// Mitsubishi GX Works2 project: project_main   PLC: Q02U

PROGRAM INPUT
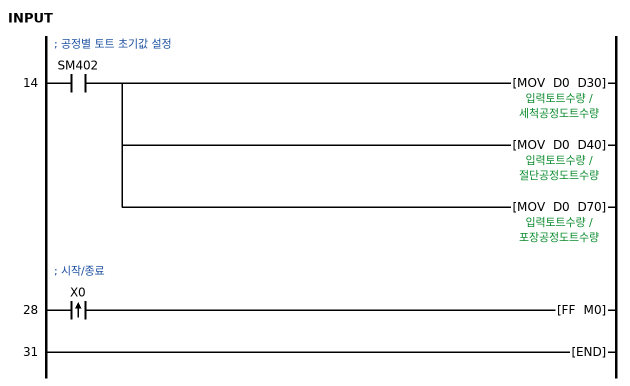
; 공정별 토트 초기값 설정
14    LD      SM402
      MOV     D0 D30  ; 입력토트수량 / 세척공정도트수량
      MOV     D0 D40  ; 절단공정도트수량
      MOV     D0 D70  ; 포장공정도트수량
; 시작/종료
28    LDP     X0
      FF      M0
31    END
END_PROGRAM

PROGRAM 세척공정
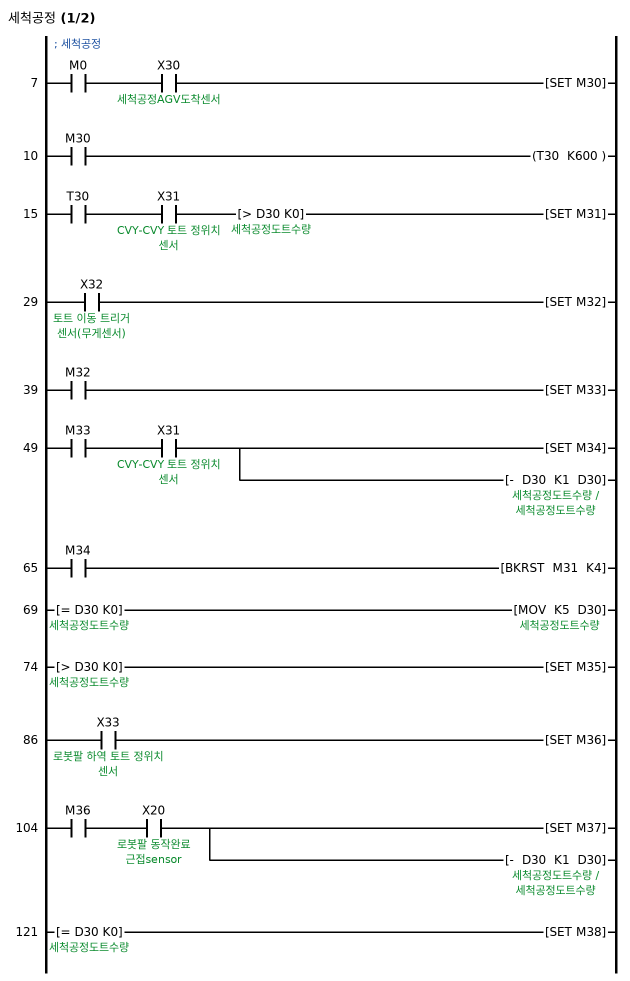
; 세척공정
7     LD      M0
      AND     X30  ; 세척공정AGV도착센서
      SET     M30
10    LD      M30
      OUT     T30 K600
15    LD      T30
      AND     X31  ; CVY-CVY 토트 정위치 센서
      AND>    D30 K0  ; 세척공정도트수량
      SET     M31
        [note] MainCVY ON
29    LD      X32  ; 토트 이동 트리거 센서(무게센서)
      SET     M32
        [note] MAinCVY OFF
39    LD      M32
      SET     M33
        [note] SubCVY1,2 ON
49    LD      M33
      AND     X31  ; CVY-CVY 토트 정위치 센서
      SET     M34
        [note] SubCVY1,2 OFF
      -       D30 K1 D30
65    LD      M34
      BKRST   M31 K4
69    LD=     D30 K0  ; 세척공정도트수량
      MOV     K5 D30
74    LD>     D30 K0  ; 세척공정도트수량
      SET     M35
        [note] SubCVY2 ON
86    LD      X33  ; 로봇팔 하역 토트 정위치 센서
      SET     M36
        [note] SubCVY2 OFF, 하역 로봇팔 ON
104   LD      M36
      AND     X20  ; 로봇팔 동작완료 근접sensor
      SET     M37
        [note] 하역 로봇팔 OFF
      -       D30 K1 D30
121   LD=     D30 K0  ; 세척공정도트수량
      SET     M38
        [note] AGV 다음 공정 이동
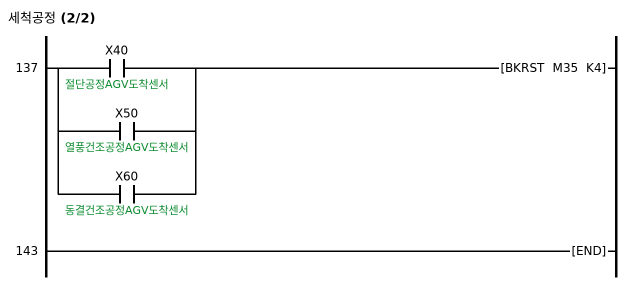
137   LD      X40  ; 절단공정AGV도착센서
      OR      X50  ; 열풍건조공정AGV도착센서
      OR      X60  ; 동결건조공정AGV도착센서
      BKRST   M35 K4
143   END
END_PROGRAM

PROGRAM 열풍건조
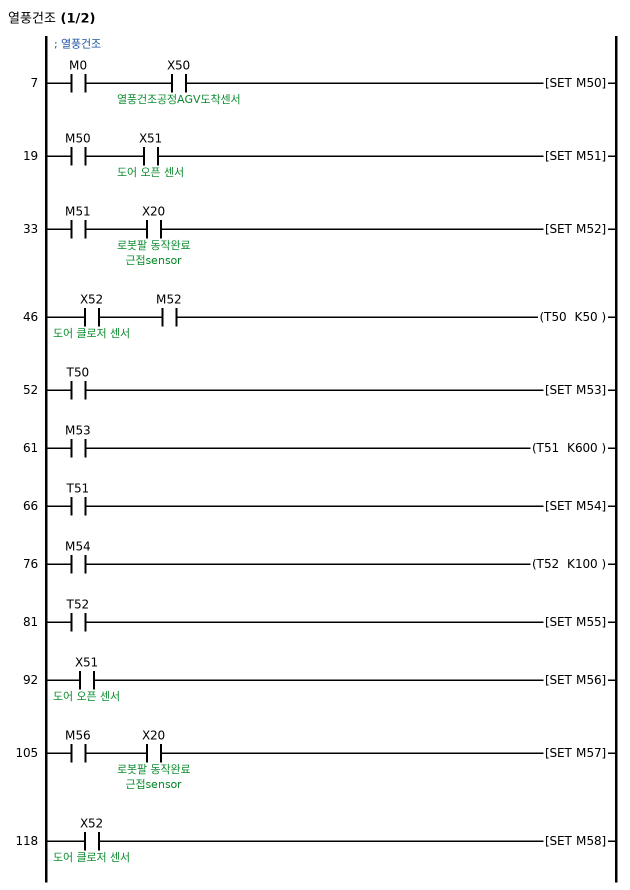
; 열풍건조
7     LD      M0
      AND     X50  ; 열풍건조공정AGV도착센서
      SET     M50
        [note] 도어 오픈CLY
19    LD      M50
      AND     X51  ; 도어 오픈 센서
      SET     M51
        [note] 상역 로봇 팔동작
33    LD      M51
      AND     X20  ; 로봇팔 동작완료 근접sensor
      SET     M52
        [note] 도어 클로즈CYL
46    LD      X52  ; 도어 클로저 센서
      AND     M52
      OUT     T50 K50
52    LD      T50
      SET     M53
        [note] 건조기 ON
61    LD      M53
      OUT     T51 K600
66    LD      T51
      SET     M54
        [note] 건조기 OFF
76    LD      M54
      OUT     T52 K100
81    LD      T52
      SET     M55
        [note] 도어 오픈CYL
92    LD      X51  ; 도어 오픈 센서
      SET     M56
        [note] 하역 로봇팔 동작
105   LD      M56
      AND     X20  ; 로봇팔 동작완료 근접sensor
      SET     M57
        [note] 도어 클로즈CYL
118   LD      X52  ; 도어 클로저 센서
      SET     M58
        [note] AGV 다음 공정 이동
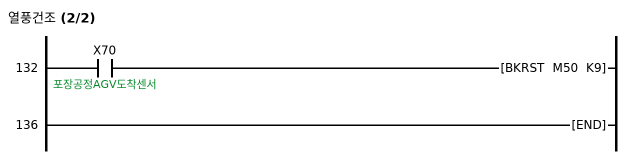
132   LD      X70  ; 포장공정AGV도착센서
      BKRST   M50 K9
136   END
END_PROGRAM

PROGRAM OUTPUT
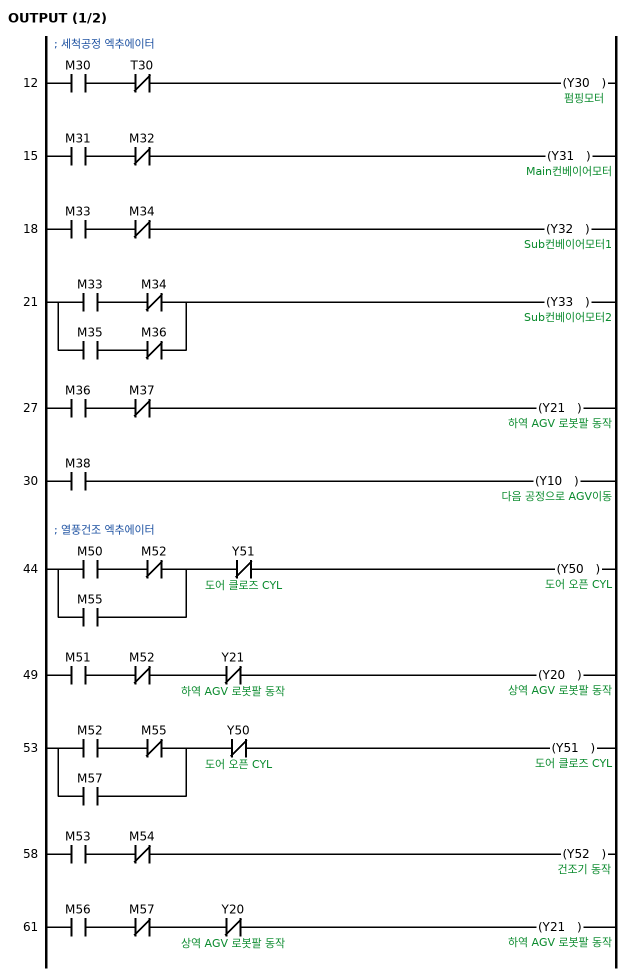
; 세척공정 엑추에이터
12    LD      M30
      ANI     T30
      OUT     Y30  ; 펌핑모터
15    LD      M31
      ANI     M32
      OUT     Y31  ; Main컨베이어모터
18    LD      M33
      ANI     M34
      OUT     Y32  ; Sub컨베이어모터1
21    LD      M33
      ANI     M34
      LD      M35
      ANI     M36
      ORB
      OUT     Y33  ; Sub컨베이어모터2
27    LD      M36
      ANI     M37
      OUT     Y21  ; 하역 AGV 로봇팔 동작
30    LD      M38
      OUT     Y10  ; 다음 공정으로 AGV이동
; 열풍건조 엑추에이터
44    LD      M50
      ANI     M52
      OR      M55
      ANI     Y51  ; 도어 클로즈 CYL
      OUT     Y50  ; 도어 오픈 CYL
49    LD      M51
      ANI     M52
      ANI     Y21  ; 하역 AGV 로봇팔 동작
      OUT     Y20  ; 상역 AGV 로봇팔 동작
53    LD      M52
      ANI     M55
      OR      M57
      ANI     Y50  ; 도어 오픈 CYL
      OUT     Y51  ; 도어 클로즈 CYL
58    LD      M53
      ANI     M54
      OUT     Y52  ; 건조기 동작
61    LD      M56
      ANI     M57
      ANI     Y20  ; 상역 AGV 로봇팔 동작
      OUT     Y21  ; 하역 AGV 로봇팔 동작
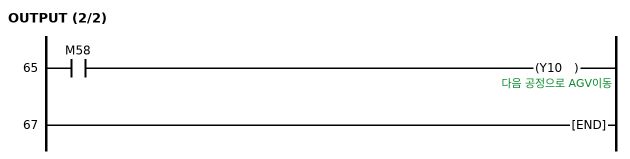
65    LD      M58
      OUT     Y10  ; 다음 공정으로 AGV이동
67    END
END_PROGRAM

// device comments not shown above
X12  ; 토틀 감지 센서
X61  ; 도어 오픈 센서
X62  ; 도어 클로저 센서
D50  ; 열풍건조공정도트수량
D60  ; 동결건조공정도트수량
